Staubli VAL3: load.pgx

public program load(string x_sItem, num& x_nResult)
  local string l_sType
  local string l_sMessage
begin
  // load the select trajectory..already loaded
  call getTrajType(l_sType)
  if find(pt:libPath(),saveData:sPathTraj)==-1
    pt:libLoad(saveData:sPathTraj+l_sType)
    delay(0)
    if saveData:bDebug
      ? "loading JPOINT..."+saveData:sPathTraj+l_sType
    endIf
  endIf
  // use the type...
  if isDefined(pt:tTraj[x_sItem])
    // use the type...
    jEditPoint=pt:tTraj[x_sItem]
    jEditPoint.sID=x_sItem
    x_nResult=0
  elseIf x_sItem!="" and find(x_sItem,"@")==-1
    // not FOUND
    call language:message(l_sMessage,-7)
    x_nResult=-1
    popUpMsg(l_sMessage+x_sItem)
    jEditPoint.sID=""
  elseIf x_sItem==""
    // reload all the template
    x_nResult=home:libLoad(saveData:sPathTraj+"HOME")
    if saveData:bDebug
      ? "loading JPOINT HOME..."+saveData:sPathTraj+"HOME"
    endIf
  endIf
end
